{attribute 'pack_mode' := '2'}
TYPE ST_FLY_CTRL :
STRUCT
  eCmd               : E_AXIS_CTRL;    // commanded axis function
END_STRUCT
END_TYPE

(* stored: Version 1.1.0.1, ProductVersion 3.1.4026.18
   DUT ST_FLY_CTRL: Id {36fad207-e492-409e-8a9f-a421a676ee20} *)
